TYPE ST120_Recipe_t :
STRUCT
    xUseVerLeft       : BOOL; // Is the left vertical picker element is used
    xUseVerRight      : BOOL; // Is the right vertical picker element is used
    FeederConfigLeft  : FeederDelays_t;
    FeederConfigRight : FeederDelays_t;
END_STRUCT
END_TYPE

(* stored: Version 1.1.0.1, ProductVersion 3.1.4024.6
   DUT ST120_Recipe_t: Id {9403bfc6-5a03-4fd8-a37a-1b19e718cfc1} *)
